Universal Robots PolyScope program: Rulleband_Robot.urp

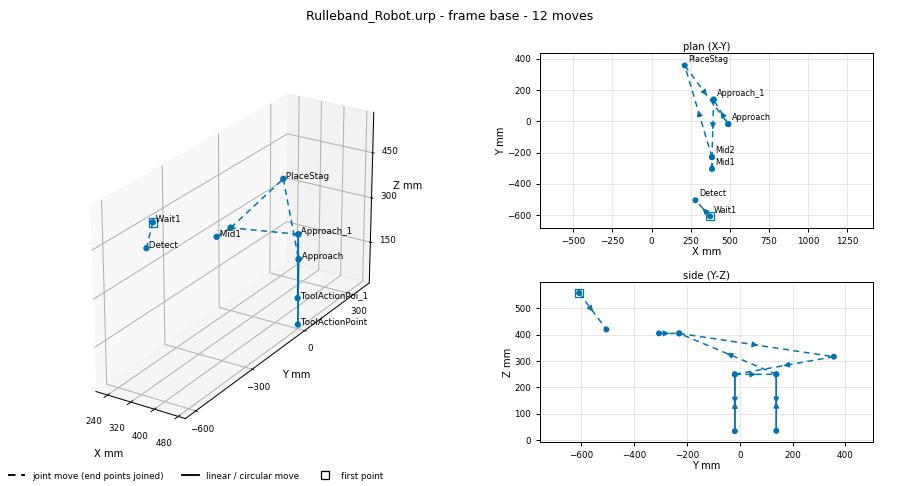
[picture p0: tool path of Rulleband_Robot.urp in frame base, 12 of 15 moves have a stored position in this frame; points joined in program order, loops and branches not executed]
Program Rulleband_Robot (installation=Rulleband directory=/programs/usbdisk createdIn=5.13.1 lastSavedIn=5.13.1 robotSerialNumber=20235501174)
Calibrated DH parameters: a=[0.000032, -0.325726, -0.190194, 0.000039, -0.000028, 0]; d=[0.162658, 160.336908, 38.259061, -198.462712, 0.099728, 0.099683]; alpha=[1.570908, 0.001706, -0.001729, 1.570164, -1.570565, 0]; deltaTheta=[0, 0.6986, 4.51965, 1.064934, 0, 0]
InitVariablesNode variables(variable(name=EyesPickAppr, expression=p[0.0,0.0,0.0,0.0,0.0,0.0]), variable(name=EyesPickPose, expression=p[0.0,0.0,0.0,0.0,0.0,0.0]), variable(name=EyesWorkpCount, expression=-1), variable(name=EyesWorkpPose, expression=p[0.0,0.0,0.0,0.0,0.0,0.0]), variable(name=EyesWorkpiece, expression=-1), variable(name=Pallet_1_lct, expression=1), variable(name=Pallet_1_lno, expression=1), variable(name=Pallet_1_sep, expression=False), variable(name=Pallet_1_tct, expression=1), variable(name=Pallet_2_lct, expression=1), variable(name=Pallet_2_lno, expression=1), variable(name=Pallet_2_sep, expression=False), variable(name=Pallet_2_tct, expression=1))
Robot Program (runOnlyOnce=false)
  Set ExpressionOutput pin=BoxPickedUp; expression=0
  MoveJ speed 60 deg/s, acceleration 80 deg/s^2 (useActiveTCP=true) feature=Base
    Waypoint Wait1: TCP in base x=374.736 y=-607.924 z=557.819 mm, rx=-1.057 ry=2.4926 rz=-1.0214 rad; joints [-47.428, -100.08, -66.805, -59.519, 89.919, -3.664] deg; TCP offset x=0 y=0 z=150.6 mm, rx=0 ry=0 rz=0 rad
  Wait DigitalInput pin=Stop; digitalValue=0
  URCap TCP (OnRobot, OnRobot A/S)
  URCap 2FG Release (OnRobot, OnRobot A/S) dataModel(external_internal_action.index=0, twofg.target-speed=50, twofg.external-grip.target-width=0.07, twofg.internal-grip.target-width=0.084)
  Wait DigitalInput pin=BoxDetected; digitalValue=1
  MoveJ speed 60 deg/s, acceleration 80 deg/s^2 (useActiveTCP=true) feature=Base
    Waypoint Detect: TCP in base x=280.612 y=-504.64 z=419.473 mm, rx=-1.2255 ry=2.886 rz=-0.0229 rad; joints [-47.445, -100.22, -66.954, -101.936, 89.93, -3.655] deg
  URCap Eyes Locate (OnRobot, OnRobot A/S) dataModel(eye-process-uid=1, eye-program-calib=0)
    URCap Eyes Get Workpiece (OnRobot, OnRobot A/S) dataModel(programTypeKey=0, programCalibTypeKey=0, countAssignmentKey=EyesWorkpCount≔eyes_workp_cnt, locatePoseAssignmentKey=EyesWorkpPose≔eyes_workp_pose, workpieceAssignmentKey=EyesWorkpiece≔eyes_workp_type, Variable(key=objCntKey, variable(name=EyesWorkpCount, initializeExpression=-1)), Variable(key=objPosKey, variable(name=EyesWorkpPose, initializeExpression=p[0.0,0.0,0.0,0.0,0.0,0.0])), Variable(key=objResKey, variable(name=EyesWorkpiece, initializeExpression=-1))); state(isChildrenLocked=true)
      EyesWorkpCount := eyes_workp_cnt
      EyesWorkpPose := eyes_workp_pose
      EyesWorkpiece := eyes_workp_type
      Folder Commands
        URCap Eyes Pick (OnRobot, OnRobot A/S) dataModel(Variable(key=eyePickApproachPoseKey, variable(name=EyesPickAppr, initializeExpression=p[0.0,0.0,0.0,0.0,0.0,0.0])), Variable(key=eyePickPoseKey, variable(name=EyesPickPose, initializeExpression=p[0.0,0.0,0.0,0.0,0.0,0.0]))); state(isChildrenLocked=true)
          URCap TCP (OnRobot, OnRobot A/S) dataModel(tool-index=1)
          MoveJ speed 60 deg/s, acceleration 80 deg/s^2 (useActiveTCP=false) tcp=OnRobot_Default; feature=Base
            Waypoint Variable (Variable): variable=EyesPickAppr
          MoveL speed 250 mm/s, acceleration 1200 mm/s^2 (useActiveTCP=false) tcp=OnRobot_Default; feature=Base
            Waypoint Variable (Variable): variable=EyesPickPose
          URCap 2FG Grip (OnRobot, OnRobot A/S) dataModel(tool-index=1, twofg.external-grip.target-width=0.045, twofg.internal-grip.target-width=0.059)
          MoveL speed 250 mm/s, acceleration 1200 mm/s^2 (useActiveTCP=false) tcp=OnRobot_Default; feature=Base
            Waypoint Variable (Variable): variable=EyesPickAppr
            MoveJ speed 60 deg/s, acceleration 80 deg/s^2 (useActiveTCP=true) feature=Base
              Waypoint Mid1: TCP in base x=386.597 y=-305.445 z=404.702 mm, rx=-2.2825 ry=2.1521 rz=-0.0214 rad; joints [-22.423, -87.843, -82.462, -98.887, 89.826, -25.978] deg
              Set ExpressionOutput pin=BoxPickedUp; expression=1
            MoveJ speed 60 deg/s, acceleration 80 deg/s^2 (useActiveTCP=true) feature=Base
              Waypoint Mid2: TCP in base x=386.595 y=-229.268 z=404.71 mm, rx=2.3979 ry=-2.0088 rz=0.045 rad; joints [-12.4, -81.391, -88.336, -99.169, 88.429, -22.684] deg
              Set ExpressionOutput pin=BoxPickedUp; expression=0
            If StackStag
              MoveJ speed 60 deg/s, acceleration 80 deg/s^2 (useActiveTCP=true) feature=Base
                Waypoint PlaceStag: TCP in base x=212.453 y=356.51 z=316.398 mm, rx=2.8842 ry=-1.2264 rz=-0.007 rad; joints [77.907, -76.807, -104.535, -89.044, 90.203, 33.794] deg
                URCap 2FG Release (OnRobot, OnRobot A/S) dataModel(external_internal_action.index=0, twofg.target-speed=50, twofg.external-grip.target-width=0.07, twofg.internal-grip.target-width=0.084)
            ElseIf StackQube
              MoveJ speed 60 deg/s, acceleration 80 deg/s^2 (useActiveTCP=true) feature=Base
                URCap Palletizing (polyscope-pallet-impl, Universal Robots) dataModel(palletFeature=Base, isPalletizing=true, rememberTraversal=true, Variable(key=layerNumberVariable, variable(name=Pallet_1_lno, initializeExpression=1)), Variable(key=layerCountingVariable, variable(name=Pallet_1_lct, initializeExpression=1)), Variable(key=handleSeparatorVariable, variable(name=Pallet_1_sep, initializeExpression=False)), Variable(key=totalCountVariable, variable(name=Pallet_1_tct, initializeExpression=1)), Variable(key=name, variable(name=PalletQube)), Length(key=objectHeight value=0.05 unit=M), Variable(key=globalCountingVariable, variable=CountCube), Variable(key=referencePoint, variable(featureName=referencePoint)), Variable(key=separatorPoint, variable(featureName=separatorPoint))); state(isChildrenLocked=true)
                  URCap Patterns (polyscope-pallet-impl, Universal Robots) state(isChildrenLocked=true)
                    URCap Pattern (polyscope-pallet-impl, Universal Robots) dataModel(UUID=3706cdfc-62e9-4a56-97f1-525e60ec2df3, patternType=GRID, rows=2, columns=2, Variable(key=nameVariable, variable(name=Grid_Pattern_1))); state(isChildrenLocked=true)
                      URCap Item (polyscope-pallet-impl, Universal Robots) dataModel(UUID=cd952b8b-bd85-4f89-a54d-d6ded2810822, patternType=GRID, index=0, calibrationDeltaTheta=[-5.619853506513839E-8, 0.6985999251272134, 4.51964984537941, 1.064933905038163, -3.8282480393017626E-7, 1.5672308527857337E-7], calibrationA=[3.240606463539282E-5, -0.3257255848617904, -0.19019392699174165, 3.918782199125579E-5, -2.84956439719103E-5, 0.0], calibrationD=[0.16265814840147477, 160.33690781595612, 38.25906128387399, -198.4627121750024, 0.09972815606269109, 0.09968261467078814], calibrationAlpha=[1.5709076652034195, 0.0017062724619852482, -0.001728875805344314, 1.570164167718445, -1.570565344071262, 0.0], calibrationJointChecksum=[-1287093867, -1288866224, 880150339, -1277156834, -1273404925, -1273938844], calibrationStatus=2, calibrationValidChecksum=true, baseToFeature=[0.0, 0.0, 0.0, 0.0, 0.0, 0.0], TCPOffset=[8.204032315717313E-6, -5.9162667255807655E-6, 0.15059004793773445, 2.4115821225276227E-5, 4.099301157486997E-5, -2.0000813522386773E-5], Variable(key=variable, variable(name=CornerItem_1)), JointPositions(key=jointpositions, JointPosition(key=[1], Angle(key=pos value=0.236204 unit=RAD)), JointPosition(key=[2], Angle(key=pos value=-1.818807 unit=RAD)), JointPosition(key=[3], Angle(key=pos value=-2.170231 unit=RAD)), JointPosition(key=[4], Angle(key=pos value=-0.68602 unit=RAD)), JointPosition(key=[5], Angle(key=pos value=1.577194 unit=RAD)), JointPosition(key=[6], Angle(key=pos value=-0.550482 unit=RAD))))
                      URCap Item (polyscope-pallet-impl, Universal Robots) dataModel(UUID=510a2751-c89f-48d7-b5ec-b82c6880e835, patternType=GRID, index=1, calibrationDeltaTheta=[-5.619853506513839E-8, 0.6985999251272134, 4.51964984537941, 1.064933905038163, -3.8282480393017626E-7, 1.5672308527857337E-7], calibrationA=[3.240606463539282E-5, -0.3257255848617904, -0.19019392699174165, 3.918782199125579E-5, -2.84956439719103E-5, 0.0], calibrationD=[0.16265814840147477, 160.33690781595612, 38.25906128387399, -198.4627121750024, 0.09972815606269109, 0.09968261467078814], calibrationAlpha=[1.5709076652034195, 0.0017062724619852482, -0.001728875805344314, 1.570164167718445, -1.570565344071262, 0.0], calibrationJointChecksum=[-1287093867, -1288866224, 880150339, -1277156834, -1273404925, -1273938844], calibrationStatus=2, calibrationValidChecksum=true, baseToFeature=[0.0, 0.0, 0.0, 0.0, 0.0, 0.0], TCPOffset=[4.739870851172556E-5, -1.39329689071932E-4, 0.15014656861322506, 0.0010031032300477248, 4.0907584354029015E-4, -1.9752972107160844E-5], Variable(key=variable, variable(name=CornerItem_2)), JointPositions(key=jointpositions, JointPosition(key=[1], Angle(key=pos value=0.368593 unit=RAD)), JointPosition(key=[2], Angle(key=pos value=-1.727822 unit=RAD)), JointPosition(key=[3], Angle(key=pos value=-2.280992 unit=RAD)), JointPosition(key=[4], Angle(key=pos value=-0.689674 unit=RAD)), JointPosition(key=[5], Angle(key=pos value=1.577764 unit=RAD)), JointPosition(key=[6], Angle(key=pos value=-0.428085 unit=RAD))))
                      URCap Item (polyscope-pallet-impl, Universal Robots) dataModel(UUID=e122b4bc-d435-4b3e-8145-a6d3b084f54d, patternType=GRID, index=2, calibrationDeltaTheta=[-5.619853506513839E-8, 0.6985999251272134, 4.51964984537941, 1.064933905038163, -3.8282480393017626E-7, 1.5672308527857337E-7], calibrationA=[3.240606463539282E-5, -0.3257255848617904, -0.19019392699174165, 3.918782199125579E-5, -2.84956439719103E-5, 0.0], calibrationD=[0.16265814840147477, 160.33690781595612, 38.25906128387399, -198.4627121750024, 0.09972815606269109, 0.09968261467078814], calibrationAlpha=[1.5709076652034195, 0.0017062724619852482, -0.001728875805344314, 1.570164167718445, -1.570565344071262, 0.0], calibrationJointChecksum=[-1287093867, -1288866224, 880150339, -1277156834, -1273404925, -1273938844], calibrationStatus=2, calibrationValidChecksum=true, baseToFeature=[0.0, 0.0, 0.0, 0.0, 0.0, 0.0], TCPOffset=[-1.302004762687714E-5, 6.1165934424622925E-6, 0.15060578596154484, 1.183214839352049E-6, -4.440827486682168E-5, 3.1158120793490084E-7], Variable(key=variable, variable(name=CornerItem_3)), JointPositions(key=jointpositions, JointPosition(key=[1], Angle(key=pos value=0.313012 unit=RAD)), JointPosition(key=[2], Angle(key=pos value=-1.636409 unit=RAD)), JointPosition(key=[3], Angle(key=pos value=-2.396776 unit=RAD)), JointPosition(key=[4], Angle(key=pos value=-0.637643 unit=RAD)), JointPosition(key=[5], Angle(key=pos value=1.573321 unit=RAD)), JointPosition(key=[6], Angle(key=pos value=-0.495543 unit=RAD))))
                      URCap Item (polyscope-pallet-impl, Universal Robots) dataModel(UUID=abdb20b7-ed23-4633-bc3e-51a6e786a5f8, patternType=GRID, index=3, calibrationDeltaTheta=[-5.619853506513839E-8, 0.6985999251272134, 4.51964984537941, 1.064933905038163, -3.8282480393017626E-7, 1.5672308527857337E-7], calibrationA=[3.240606463539282E-5, -0.3257255848617904, -0.19019392699174165, 3.918782199125579E-5, -2.84956439719103E-5, 0.0], calibrationD=[0.16265814840147477, 160.33690781595612, 38.25906128387399, -198.4627121750024, 0.09972815606269109, 0.09968261467078814], calibrationAlpha=[1.5709076652034195, 0.0017062724619852482, -0.001728875805344314, 1.570164167718445, -1.570565344071262, 0.0], calibrationJointChecksum=[-1287093867, -1288866224, 880150339, -1277156834, -1273404925, -1273938844], calibrationStatus=2, calibrationValidChecksum=true, baseToFeature=[0.0, 0.0, 0.0, 0.0, 0.0, 0.0], TCPOffset=[4.8950441163264635E-6, -8.673804605618951E-6, 0.15059616075054685, -4.510320043319502E-6, 3.9076449391734386E-5, -1.0625925758525127E-5], Variable(key=variable, variable(name=CornerItem_4)), JointPositions(key=jointpositions, JointPosition(key=[1], Angle(key=pos value=0.188671 unit=RAD)), JointPosition(key=[2], Angle(key=pos value=-1.756131 unit=RAD)), JointPosition(key=[3], Angle(key=pos value=-2.241869 unit=RAD)), JointPosition(key=[4], Angle(key=pos value=-0.706567 unit=RAD)), JointPosition(key=[5], Angle(key=pos value=1.547311 unit=RAD)), JointPosition(key=[6], Angle(key=pos value=-0.629233 unit=RAD))))
                  URCap Layers (polyscope-pallet-impl, Universal Robots) dataModel(separators=[false, false, false], selectedPatterns=[3706cdfc-62e9-4a56-97f1-525e60ec2df3, 3706cdfc-62e9-4a56-97f1-525e60ec2df3, 3706cdfc-62e9-4a56-97f1-525e60ec2df3])
                  URCap At Each Item (polyscope-pallet-impl, Universal Robots) dataModel(selectedPattern=3706cdfc-62e9-4a56-97f1-525e60ec2df3, selectedPosition=cd952b8b-bd85-4f89-a54d-d6ded2810822, Approach_calibrationDeltaTheta=[-5.619853506513839E-8, 0.6985999251272134, 4.51964984537941, 1.064933905038163, -3.8282480393017626E-7, 1.5672308527857337E-7], Approach_calibrationA=[3.240606463539282E-5, -0.3257255848617904, -0.19019392699174165, 3.918782199125579E-5, -2.84956439719103E-5, 0.0], Approach_calibrationD=[0.16265814840147477, 160.33690781595612, 38.25906128387399, -198.4627121750024, 0.09972815606269109, 0.09968261467078814], Approach_calibrationAlpha=[1.5709076652034195, 0.0017062724619852482, -0.001728875805344314, 1.570164167718445, -1.570565344071262, 0.0], Approach_calibrationJointChecksum=[-1287093867, -1288866224, 880150339, -1277156834, -1273404925, -1273938844], Approach_calibrationStatus=2, Approach_calibrationValidChecksum=true, Approach_baseToFeature=[0.0, 0.0, 0.0, 0.0, 0.0, 0.0], Approach_TCPOffset=[-2.484949580883189E-6, -5.889260084268599E-6, 0.15060151156702636, 7.514828417656885E-6, -1.7652884040941386E-5, 1.1806071274247617E-5], Exit_calibrationDeltaTheta=[-5.619853506513839E-8, 0.6985999251272134, 4.51964984537941, 1.064933905038163, -3.8282480393017626E-7, 1.5672308527857337E-7], Exit_calibrationA=[3.240606463539282E-5, -0.3257255848617904, -0.19019392699174165, 3.918782199125579E-5, -2.84956439719103E-5, 0.0], Exit_calibrationD=[0.16265814840147477, 160.33690781595612, 38.25906128387399, -198.4627121750024, 0.09972815606269109, 0.09968261467078814], Exit_calibrationAlpha=[1.5709076652034195, 0.0017062724619852482, -0.001728875805344314, 1.570164167718445, -1.570565344071262, 0.0], Exit_calibrationJointChecksum=[-1287093867, -1288866224, 880150339, -1277156834, -1273404925, -1273938844], Exit_calibrationStatus=2, Exit_calibrationValidChecksum=true, Exit_baseToFeature=[0.0, 0.0, 0.0, 0.0, 0.0, 0.0], Exit_TCPOffset=[-5.265586045133386E-6, -3.0020935677388394E-6, 0.15061823806701954, -3.9875281205960976E-5, -2.2872559796053934E-5, -4.3081602447660284E-5], currentWizardState=LANDING, Pose(key=refBaseToFeature, Position(key=posePosition, Length(key=X value=0 unit=M), Length(key=Y value=0 unit=M), Length(key=Z value=0 unit=M)), Rotation(key=poseRotation, Angle(key=RX value=0 unit=RAD), Angle(key=RY value=0 unit=RAD), Angle(key=RZ value=0 unit=RAD))), Pose(key=refPose, Position(key=posePosition, Length(key=X value=0.490821 unit=M), Length(key=Y value=-0.018345 unit=M), Length(key=Z value=0.034429 unit=M)), Rotation(key=poseRotation, Angle(key=RX value=-2.875425 unit=RAD), Angle(key=RY value=1.195044 unit=RAD), Angle(key=RZ value=-0.041344 unit=RAD))), JointPositions(key=Approach_jointpositions, JointPosition(key=[1], Angle(key=pos value=0.236641 unit=RAD)), JointPosition(key=[2], Angle(key=pos value=-1.529418 unit=RAD)), JointPosition(key=[3], Angle(key=pos value=-1.847126 unit=RAD)), JointPosition(key=[4], Angle(key=pos value=-1.298465 unit=RAD)), JointPosition(key=[5], Angle(key=pos value=1.575698 unit=RAD)), JointPosition(key=[6], Angle(key=pos value=-0.54988 unit=RAD))), JointPositions(key=Exit_jointpositions, JointPosition(key=[1], Angle(key=pos value=0.236641 unit=RAD)), JointPosition(key=[2], Angle(key=pos value=-1.529593 unit=RAD)), JointPosition(key=[3], Angle(key=pos value=-1.847763 unit=RAD)), JointPosition(key=[4], Angle(key=pos value=-1.297653 unit=RAD)), JointPosition(key=[5], Angle(key=pos value=1.575699 unit=RAD)), JointPosition(key=[6], Angle(key=pos value=-0.549881 unit=RAD))))
                    URCap Generated Movements (polyscope-pallet-impl, Universal Robots) state(isChildrenLocked=true)
                      MoveJ speed 60 deg/s, acceleration 80 deg/s^2 (useActiveTCP=true) feature=referencePoint
                        Waypoint Approach: TCP in base x=490.824 y=-18.339 z=249.726 mm, rx=-2.8754 ry=1.1951 rz=-0.0413 rad; joints [13.559, -87.629, -105.833, -74.397, 90.281, -31.506] deg; TCP offset x=-0.002 y=-0.006 z=150.602 mm, rx=0 ry=0 rz=0 rad; feature pose in base x=490.821 y=-18.345 z=34.429 mm, rx=-2.8754 ry=1.195 rz=-0.0413 rad
                      MoveL speed 250 mm/s, acceleration 1200 mm/s^2 (useActiveTCP=true) feature(featureName=referencePoint)
                        Waypoint ToolActionPoint: TCP in base x=490.821 y=-18.345 z=34.429 mm, rx=-2.8754 ry=1.195 rz=-0.0413 rad; joints [13.534, -104.21, -124.345, -39.306, 90.367, -31.54] deg; TCP offset x=0.008 y=-0.006 z=150.59 mm, rx=0 ry=0 rz=0 rad
                      Folder Tool action
                        URCap 2FG Release (OnRobot, OnRobot A/S) dataModel(external_internal_action.index=0, twofg.target-speed=50, twofg.external-grip.target-width=0.07, twofg.internal-grip.target-width=0.084)
                      MoveL speed 250 mm/s, acceleration 1200 mm/s^2 (useActiveTCP=true) feature(featureName=referencePoint)
                        Waypoint Exit_1: TCP in base x=490.82 y=-18.339 z=249.403 mm, rx=-2.8755 ry=1.195 rz=-0.0413 rad; joints [13.559, -87.639, -105.869, -74.35, 90.281, -31.506] deg; TCP offset x=-0.005 y=-0.003 z=150.618 mm, rx=0 ry=0 rz=0 rad
            ElseIf StackLine
              MoveJ speed 60 deg/s, acceleration 80 deg/s^2 (useActiveTCP=true) feature=Base
                URCap Palletizing (polyscope-pallet-impl, Universal Robots) dataModel(palletFeature=Base, isPalletizing=true, rememberTraversal=true, Length(key=objectHeight value=0.05 unit=M), Variable(key=name, variable(name=PalletLine)), Variable(key=globalCountingVariable, variable=CountLine), Variable(key=layerCountingVariable, variable(name=Pallet_2_lct, initializeExpression=1)), Variable(key=layerNumberVariable, variable(name=Pallet_2_lno, initializeExpression=1)), Variable(key=handleSeparatorVariable, variable(name=Pallet_2_sep, initializeExpression=False)), Variable(key=totalCountVariable, variable(name=Pallet_2_tct, initializeExpression=1)), Variable(key=referencePoint, variable(featureName=referencePoin_2)), Variable(key=separatorPoint, variable(featureName=separatorPoin_2))); state(isChildrenLocked=true)
                  URCap Patterns (polyscope-pallet-impl, Universal Robots) state(isChildrenLocked=true)
                    URCap Pattern (polyscope-pallet-impl, Universal Robots) dataModel(UUID=6d97de25-7160-4b60-982b-5d07011afd31, patternType=LINE, objects=3, Variable(key=nameVariable, variable(name=Line_Pattern_1))); state(isChildrenLocked=true)
                      URCap Item (polyscope-pallet-impl, Universal Robots) dataModel(UUID=36d71b64-4a64-4360-9de9-7a224c84a0ec, patternType=LINE, index=0, calibrationDeltaTheta=[-5.619853506513839E-8, 0.6985999251272134, 4.51964984537941, 1.064933905038163, -3.8282480393017626E-7, 1.5672308527857337E-7], calibrationA=[3.240606463539282E-5, -0.3257255848617904, -0.19019392699174165, 3.918782199125579E-5, -2.84956439719103E-5, 0.0], calibrationD=[0.16265814840147477, 160.33690781595612, 38.25906128387399, -198.4627121750024, 0.09972815606269109, 0.09968261467078814], calibrationAlpha=[1.5709076652034195, 0.0017062724619852482, -0.001728875805344314, 1.570164167718445, -1.570565344071262, 0.0], calibrationJointChecksum=[-1287093867, -1288866224, 880150339, -1277156834, -1273404925, -1273938844], calibrationStatus=2, calibrationValidChecksum=true, baseToFeature=[0.0, 0.0, 0.0, 0.0, 0.0, 0.0], TCPOffset=[-3.078339609885461E-7, -9.079620647556297E-7, 0.1506011472334898, 2.1306288581442538E-5, 1.4482090641716807E-5, 3.315399414126542E-6], Variable(key=variable, variable(name=StartItem_1)), JointPositions(key=jointpositions, JointPosition(key=[1], Angle(key=pos value=0.661205 unit=RAD)), JointPosition(key=[2], Angle(key=pos value=-1.684585 unit=RAD)), JointPosition(key=[3], Angle(key=pos value=-2.31512 unit=RAD)), JointPosition(key=[4], Angle(key=pos value=-0.736077 unit=RAD)), JointPosition(key=[5], Angle(key=pos value=1.568725 unit=RAD)), JointPosition(key=[6], Angle(key=pos value=1.446206 unit=RAD))))
                      URCap Item (polyscope-pallet-impl, Universal Robots) dataModel(UUID=18b5165f-d4d1-40fc-b9ca-faba2c626a37, patternType=LINE, index=1, calibrationDeltaTheta=[-5.619853506513839E-8, 0.6985999251272134, 4.51964984537941, 1.064933905038163, -3.8282480393017626E-7, 1.5672308527857337E-7], calibrationA=[3.240606463539282E-5, -0.3257255848617904, -0.19019392699174165, 3.918782199125579E-5, -2.84956439719103E-5, 0.0], calibrationD=[0.16265814840147477, 160.33690781595612, 38.25906128387399, -198.4627121750024, 0.09972815606269109, 0.09968261467078814], calibrationAlpha=[1.5709076652034195, 0.0017062724619852482, -0.001728875805344314, 1.570164167718445, -1.570565344071262, 0.0], calibrationJointChecksum=[-1287093867, -1288866224, 880150339, -1277156834, -1273404925, -1273938844], calibrationStatus=2, calibrationValidChecksum=true, baseToFeature=[0.0, 0.0, 0.0, 0.0, 0.0, 0.0], TCPOffset=[-3.7644409823012204E-5, 1.0668156779053417E-5, 0.15056873189981032, -3.313694711361767E-5, -9.620511909828327E-5, 1.2540541776327372E-5], Variable(key=variable, variable(name=EndItem_1)), JointPositions(key=jointpositions, JointPosition(key=[1], Angle(key=pos value=0.988627 unit=RAD)), JointPosition(key=[2], Angle(key=pos value=-1.594005 unit=RAD)), JointPosition(key=[3], Angle(key=pos value=-2.422702 unit=RAD)), JointPosition(key=[4], Angle(key=pos value=-0.705728 unit=RAD)), JointPosition(key=[5], Angle(key=pos value=1.554927 unit=RAD)), JointPosition(key=[6], Angle(key=pos value=1.794493 unit=RAD))))
                  URCap Layers (polyscope-pallet-impl, Universal Robots) dataModel(separators=[false, false, false], selectedPatterns=[6d97de25-7160-4b60-982b-5d07011afd31, 6d97de25-7160-4b60-982b-5d07011afd31, 6d97de25-7160-4b60-982b-5d07011afd31])
                  URCap At Each Item (polyscope-pallet-impl, Universal Robots) dataModel(selectedPattern=6d97de25-7160-4b60-982b-5d07011afd31, selectedPosition=36d71b64-4a64-4360-9de9-7a224c84a0ec, Approach_calibrationDeltaTheta=[-5.619853506513839E-8, 0.6985999251272134, 4.51964984537941, 1.064933905038163, -3.8282480393017626E-7, 1.5672308527857337E-7], Approach_calibrationA=[3.240606463539282E-5, -0.3257255848617904, -0.19019392699174165, 3.918782199125579E-5, -2.84956439719103E-5, 0.0], Approach_calibrationD=[0.16265814840147477, 160.33690781595612, 38.25906128387399, -198.4627121750024, 0.09972815606269109, 0.09968261467078814], Approach_calibrationAlpha=[1.5709076652034195, 0.0017062724619852482, -0.001728875805344314, 1.570164167718445, -1.570565344071262, 0.0], Approach_calibrationJointChecksum=[-1287093867, -1288866224, 880150339, -1277156834, -1273404925, -1273938844], Approach_calibrationStatus=2, Approach_calibrationValidChecksum=true, Approach_baseToFeature=[0.0, 0.0, 0.0, 0.0, 0.0, 0.0], Approach_TCPOffset=[2.2911913218903734E-6, -4.857193455082287E-6, 0.15059645614130168, 5.374759504075437E-6, -2.1003169953275386E-5, 1.0819420624801368E-5], Exit_calibrationDeltaTheta=[-5.619853506513839E-8, 0.6985999251272134, 4.51964984537941, 1.064933905038163, -3.8282480393017626E-7, 1.5672308527857337E-7], Exit_calibrationA=[3.240606463539282E-5, -0.3257255848617904, -0.19019392699174165, 3.918782199125579E-5, -2.84956439719103E-5, 0.0], Exit_calibrationD=[0.16265814840147477, 160.33690781595612, 38.25906128387399, -198.4627121750024, 0.09972815606269109, 0.09968261467078814], Exit_calibrationAlpha=[1.5709076652034195, 0.0017062724619852482, -0.001728875805344314, 1.570164167718445, -1.570565344071262, 0.0], Exit_calibrationJointChecksum=[-1287093867, -1288866224, 880150339, -1277156834, -1273404925, -1273938844], Exit_calibrationStatus=2, Exit_calibrationValidChecksum=true, Exit_baseToFeature=[0.0, 0.0, 0.0, 0.0, 0.0, 0.0], Exit_TCPOffset=[6.255682426514753E-7, -1.3642395849750022E-5, 0.1506014118645011, 1.7150782775851313E-5, -1.3419976765097327E-7, 3.3933520228728994E-5], currentWizardState=SHOW_DONE, Pose(key=refBaseToFeature, Position(key=posePosition, Length(key=X value=0 unit=M), Length(key=Y value=0 unit=M), Length(key=Z value=0 unit=M)), Rotation(key=poseRotation, Angle(key=RX value=0 unit=RAD), Angle(key=RY value=0 unit=RAD), Angle(key=RZ value=0 unit=RAD))), Pose(key=refPose, Position(key=posePosition, Length(key=X value=0.397157 unit=M), Length(key=Y value=0.138449 unit=M), Length(key=Z value=0.035734 unit=M)), Rotation(key=poseRotation, Angle(key=RX value=1.189145 unit=RAD), Angle(key=RY value=-2.884114 unit=RAD), Angle(key=RZ value=0.012008 unit=RAD))), JointPositions(key=Approach_jointpositions, JointPosition(key=[1], Angle(key=pos value=0.661747 unit=RAD)), JointPosition(key=[2], Angle(key=pos value=-1.381902 unit=RAD)), JointPosition(key=[3], Angle(key=pos value=-1.959388 unit=RAD)), JointPosition(key=[4], Angle(key=pos value=-1.394504 unit=RAD)), JointPosition(key=[5], Angle(key=pos value=1.567224 unit=RAD)), JointPosition(key=[6], Angle(key=pos value=1.447106 unit=RAD))), JointPositions(key=Exit_jointpositions, JointPosition(key=[1], Angle(key=pos value=0.661748 unit=RAD)), JointPosition(key=[2], Angle(key=pos value=-1.381797 unit=RAD)), JointPosition(key=[3], Angle(key=pos value=-1.958932 unit=RAD)), JointPosition(key=[4], Angle(key=pos value=-1.395064 unit=RAD)), JointPosition(key=[5], Angle(key=pos value=1.567223 unit=RAD)), JointPosition(key=[6], Angle(key=pos value=1.447108 unit=RAD))))
                    URCap Generated Movements (polyscope-pallet-impl, Universal Robots) state(isChildrenLocked=true)
                      MoveJ speed 60 deg/s, acceleration 80 deg/s^2 (useActiveTCP=true) feature=referencePoin_2
                        Waypoint Approach_1: TCP in base x=397.159 y=138.444 z=249.834 mm, rx=1.1891 ry=-2.8841 rz=0.012 rad; joints [37.915, -79.177, -112.265, -79.899, 89.795, 82.913] deg; TCP offset x=0.002 y=-0.005 z=150.596 mm, rx=0 ry=0 rz=0 rad; feature pose in base x=397.157 y=138.449 z=35.734 mm, rx=1.1891 ry=-2.8841 rz=0.012 rad
                      MoveL speed 250 mm/s, acceleration 1200 mm/s^2 (useActiveTCP=true) feature(featureName=referencePoin_2)
                        Waypoint ToolActionPoi_1: TCP in base x=397.157 y=138.449 z=35.734 mm, rx=1.1891 ry=-2.8841 rz=0.012 rad; joints [37.884, -96.52, -132.647, -42.174, 89.881, 82.862] deg; TCP offset x=0 y=-0.001 z=150.601 mm, rx=0 ry=0 rz=0 rad
                      Folder Tool action
                        URCap 2FG Release (OnRobot, OnRobot A/S) dataModel(external_internal_action.index=0, twofg.target-speed=50, twofg.external-grip.target-width=0.07, twofg.internal-grip.target-width=0.084)
                      MoveL speed 250 mm/s, acceleration 1200 mm/s^2 (useActiveTCP=true) feature(featureName=referencePoin_2)
                        Waypoint Exit_2: TCP in base x=397.166 y=138.439 z=250.036 mm, rx=1.1891 ry=-2.8841 rz=0.012 rad; joints [37.915, -79.171, -112.239, -79.931, 89.795, 82.913] deg; TCP offset x=0.001 y=-0.014 z=150.601 mm, rx=0 ry=0 rz=0 rad
            MoveJ speed 60 deg/s, acceleration 80 deg/s^2 (useActiveTCP=true) feature=Base
              Waypoint Mid2: TCP in base x=386.595 y=-229.268 z=404.71 mm, rx=2.3979 ry=-2.0088 rz=0.045 rad; joints [-12.4, -81.391, -88.336, -99.169, 88.429, -22.684] deg; TCP offset x=0 y=0 z=150.6 mm, rx=0 ry=0 rz=0 rad
Thread Thread_2 (runOnlyOnce=false)
  If ResetQube
    Script: CountCube=0
  If ResetLine
    Script: CountLine=0
  Wait Sleep waitTime=0.01
